FUNCTION_BLOCK PnpXYCalculatorBA (* Composite Function Block Type *)
  (* Standard: 61499-2 *)
  (* Version 0.2, 2003-12-05, JHC, Rockwell Automation, Renamed from NEWCOMPFB. *)
  (* Version 0.1, 2002-01-08, JHC, Rockwell Automation, Added DLY FB as example. *)
  (* Version 0.0, 2000-05-27, JHC, Rockwell Automation *)
  (* Compiler header: package fb.rt.pnp; *)
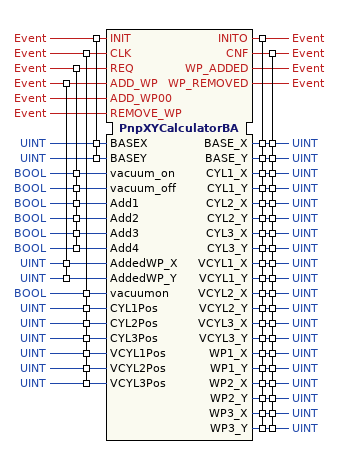
  EVENT_INPUT
    INIT WITH BASEX, BASEY; (* Initialization Request *)
    CLK WITH vacuumon, CYL1Pos, CYL2Pos, CYL3Pos, VCYL1Pos, VCYL2Pos, VCYL3Pos; (* Clock *)
    REQ WITH vacuum_on, vacuum_off, Add1, Add2, Add3, Add4;
    ADD_WP WITH AddedWP_X, AddedWP_Y;
    ADD_WP00;
    REMOVE_WP;
  END_EVENT
  EVENT_OUTPUT
    INITO WITH CYL1_X, CYL1_Y, BASE_Y, BASE_X, CYL2_X, CYL2_Y, VCYL1_X, VCYL1_Y, WP1_X, WP1_Y, WP2_X, WP2_Y, WP3_X, WP3_Y, CYL3_X, CYL3_Y, VCYL2_X, VCYL2_Y, VCYL3_X, VCYL3_Y; (* Initialization Confirm *)
    CNF WITH CYL1_X, CYL1_Y, BASE_Y, BASE_X, CYL2_X, CYL2_Y, VCYL1_X, VCYL1_Y, WP1_X, WP1_Y, WP2_X, WP2_Y, WP3_X, WP3_Y, CYL3_X, CYL3_Y, VCYL2_X, VCYL2_Y, VCYL3_X, VCYL3_Y;
    WP_ADDED;
    WP_REMOVED;
  END_EVENT
  VAR_INPUT
    BASEX : UINT;
    BASEY : UINT;
    vacuum_on : BOOL;
    vacuum_off : BOOL;
    Add1 : BOOL;
    Add2 : BOOL;
    Add3 : BOOL;
    Add4 : BOOL;
    AddedWP_X : UINT;
    AddedWP_Y : UINT;
    vacuumon : BOOL;
    CYL1Pos : UINT;
    CYL2Pos : UINT;
    CYL3Pos : UINT;
    VCYL1Pos : UINT;
    VCYL2Pos : UINT;
    VCYL3Pos : UINT;
  END_VAR
  VAR_OUTPUT
    BASE_X : UINT; (* Response Data from Socket *)
    BASE_Y : UINT; (* Response Data from Socket *)
    CYL1_X : UINT; (* Response Data from Socket *)
    CYL1_Y : UINT; (* Response Data from Socket *)
    CYL2_X : UINT; (* Response Data from Socket *)
    CYL2_Y : UINT; (* Response Data from Socket *)
    CYL3_X : UINT; (* Response Data from Socket *)
    CYL3_Y : UINT; (* Response Data from Socket *)
    VCYL1_X : UINT; (* Response Data from Socket *)
    VCYL1_Y : UINT; (* Response Data from Socket *)
    VCYL2_X : UINT; (* Response Data from Socket *)
    VCYL2_Y : UINT; (* Response Data from Socket *)
    VCYL3_X : UINT; (* Response Data from Socket *)
    VCYL3_Y : UINT; (* Response Data from Socket *)
    WP1_X : UINT; (* Response Data from Socket *)
    WP1_Y : UINT; (* Response Data from Socket *)
    WP2_X : UINT; (* Response Data from Socket *)
    WP2_Y : UINT; (* Response Data from Socket *)
    WP3_X : UINT; (* Response Data from Socket *)
    WP3_Y : UINT; (* Response Data from Socket *)
  END_VAR
  VAR
    cyl1x : UINT;
    cyl2x : UINT;
    cyl3x : UINT;
    vcyl1y : UINT;
    vcyl2y : UINT;
    vcyl3y : UINT;
    wp1x : UINT;
    wp1y : UINT;
    wp2x : UINT;
    wp2y : UINT;
    wp3x : UINT;
    wp3y : UINT;
    wp4x : UINT;
    wp4y : UINT;
    slider1 : BOOL;
    slider2 : BOOL;
    slider3 : BOOL;
    slider4 : BOOL;
    wp1on : BOOL;
    wp2on : BOOL;
    wp3on : BOOL;
    wp4on : BOOL;
  END_VAR
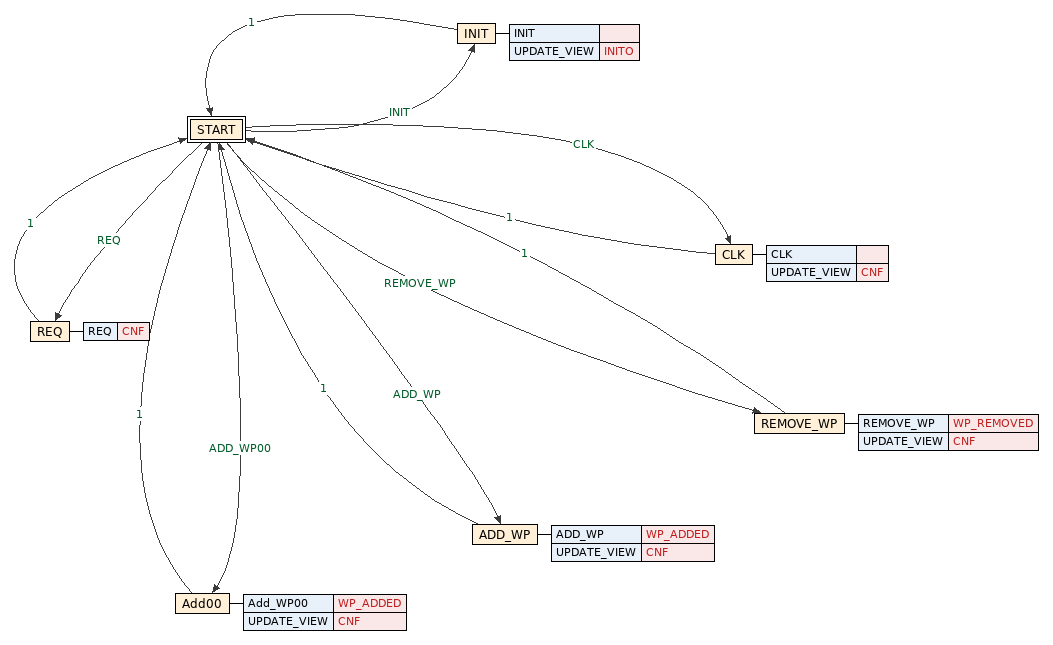
  EC_STATES
    START; (* Initial State *)
    INIT : INIT, UPDATE_VIEW -> INITO; (* Initialization *)
    REQ : REQ -> CNF; (* Normal execution *)
    CLK : CLK, UPDATE_VIEW -> CNF;
    ADD_WP : ADD_WP -> WP_ADDED, UPDATE_VIEW -> CNF;
    REMOVE_WP : REMOVE_WP -> WP_REMOVED, UPDATE_VIEW -> CNF;
    Add00 : Add_WP00 -> WP_ADDED, UPDATE_VIEW -> CNF;
  END_STATES
  EC_TRANSITIONS
    START TO INIT := INIT;
    INIT TO START := 1;
    START TO REQ := REQ;
    REQ TO START := 1;
    START TO CLK := CLK;
    CLK TO START := 1;
    START TO ADD_WP := ADD_WP;
    ADD_WP TO START := 1;
    START TO REMOVE_WP := REMOVE_WP;
    REMOVE_WP TO START := 1;
    START TO Add00 := ADD_WP00;
    Add00 TO START := 1;
  END_TRANSITIONS
  ALGORITHM INIT IN Java: (* Initialization algorithm *)
wp1x.value = 6000;
wp1y.value = 6000;
wp2x.value = 6000;
wp2y.value = 6000;
wp3x.value = 6000;
wp3y.value = 6000;
wp1on.value = false;
wp2on.value = false;
wp3on.value = false;

BASE_X.value = BASEX.value;
BASE_Y.value = BASEY.value;
CYL1_Y.value = BASEY.value;
CYL2_Y.value = BASEY.value;
CYL3_Y.value = BASEY.value;
  END_ALGORITHM
  ALGORITHM REQ IN Java: (* Normally executed algorithm *)

  END_ALGORITHM
  ALGORITHM CLK IN Java:
int cyl1_length = 75;
int cyl2_length = 75;
int cyl3_length = 150;
int vcyl1_length = 75;
int vcyl2_length = 75;
int vcyl3_length = 75;

cyl1x.value = CYL1Pos.value;
cyl2x.value = CYL2Pos.value;
cyl3x.value = CYL3Pos.value;
vcyl1y.value = VCYL1Pos.value;
vcyl2y.value = VCYL2Pos.value;
vcyl3y.value = VCYL3Pos.value;

if(WP1_X.value<=465 && WP1_Y.value>=370){
slider1.value=true;
} else {slider1.value=false;}
if(WP2_X.value<=465 && WP2_Y.value>=370){
slider2.value=true;
} else {slider2.value=false;}
if(WP3_X.value<=465 && WP3_Y.value>=370){
slider3.value=true;
} else {slider3.value=false;}


if (vacuumon.value) {
int vacuumx = VCYL3_X.value;
int vacuumy = VCYL3_Y.value+100;
int dx1 = Math.abs(wp1x.value - vacuumx);
int dy1 = Math.abs(wp1y.value - vacuumy);
int dx2 = Math.abs(wp2x.value - vacuumx);
int dy2 = Math.abs(wp2y.value - vacuumy);
int dx3 = Math.abs(wp3x.value - vacuumx);
int dy3 = Math.abs(wp3y.value - vacuumy);

if (dx1 < 17 && dy1 < 7 && wp2on.value==false && wp3on.value==false){
wp1on.value = true;
}
if (dx2 < 17 && dy2 < 7 && wp1on.value==false && wp3on.value==false){
wp2on.value = true;
}
if (dx3 < 17 && dy3 < 7 && wp2on.value==false && wp1on.value==false){
wp3on.value = true;
}
//System.out.println("Clocking"+dx1+"-"+dy1);

} else {
wp1on.value = false;
wp2on.value = false;
wp3on.value = false;
}

//System.out.println("Clocking");
  END_ALGORITHM
  ALGORITHM UPDATE_VIEW IN Java:
int bx = BASEX.value;
int by = BASEY.value;
CYL1_X.value = bx+22+cyl1x.value;
CYL2_X.value = CYL1_X.value+90+cyl2x.value;
CYL3_X.value = CYL2_X.value+90+cyl3x.value;

VCYL1_X.value = CYL3_X.value+180;
VCYL2_X.value = CYL3_X.value+180;
VCYL3_X.value = CYL3_X.value+180;
//VCYL1_Y.value = by+vcyl1y.value+15;
VCYL1_Y.value = by+vcyl1y.value;
VCYL2_Y.value = VCYL1_Y.value+90+vcyl2y.value;
VCYL3_Y.value = VCYL2_Y.value+90+vcyl3y.value;

if (wp1on.value){
wp1x.value = VCYL3_X.value;
wp1y.value = VCYL3_Y.value+100;
} else if (slider1.value){


/*if(wp1y.value <= 490) {
wp1y.value = wp1y.value+1;
if (slider2.value && wp2y.value >= 476 && wp1y.value >= 476) {
wp1y.value = wp1y.value-1;
} else if (slider3.value && wp3y.value >= 476 && wp1y.value >= 476) {
wp1y.value = wp1y.value-1;
} else if (slider3.value && slider2.value && wp2y.value >= 462 && wp3y.value >= 462 && wp1y.value >= 460) {
wp1y.value = wp1y.value-1;
}
}*/
wp1y.value = wp1y.value+1;

} else {
//wp1y.value = 385;
}

if (wp2on.value){
wp2x.value = VCYL3_X.value;
wp2y.value = VCYL3_Y.value+100;
} else if (slider2.value){



/*if(wp2y.value <= 490) {

wp2y.value = wp2y.value+1;
if (slider1.value && wp1y.value >= 476 && wp2y.value >= 476) {
wp2y.value = wp2y.value-1;
} else if (slider3.value && wp3y.value >= 476 && wp2y.value >= 476) {
wp2y.value = wp2y.value-1;
} else if (slider3.value && slider1.value && wp1y.value >= 462 && wp3y.value >= 462 && wp2y.value >= 460) {
wp2y.value = wp2y.value-1;
}

}*/
wp2y.value = wp2y.value+1;

} else {
//wp2y.value = 535;
}

if (wp3on.value){
wp3x.value = VCYL3_X.value;
wp3y.value = VCYL3_Y.value+100;
} else if (slider3.value){

/*if(wp3y.value <= 490) {

wp3y.value = wp3y.value+1;
if (slider1.value && wp1y.value >= 476 && wp3y.value >= 476) {
wp3y.value = wp3y.value-1;
} else if (slider2.value && wp2y.value >= 476 && wp3y.value >= 476) {
wp3y.value = wp3y.value-1;
} else if (slider2.value && slider1.value && wp1y.value >= 462 && wp2y.value >= 462 && wp3y.value >= 460) {
wp3y.value = wp3y.value-1;
}

}*/
wp3y.value = wp3y.value+1;


} else {
//wp3y.value = 460;
}



WP1_X.value = wp1x.value;
WP1_Y.value = wp1y.value;
WP2_X.value = wp2x.value;
WP2_Y.value = wp2y.value;
WP3_X.value = wp3x.value;
WP3_Y.value = wp3y.value;

//WP1_X.value = bx+300+wp1x.value;
WP1_Y.value = wp1y.value;
//WP2_X.value = bx+300+wp2x.value;
WP2_Y.value = wp2y.value;
//WP3_X.value = bx+300+wp3x.value;
WP3_Y.value = wp3y.value;


/*if (WP1_X.value == 462 && WP1_Y.value >= 535)
{
    WP1_X.value = 6000;
    WP1_Y.value = 6000;
}
if (WP2_X.value == 462 && WP2_Y.value >= 535)
{
    WP2_X.value = 6000;
    WP2_Y.value = 6000;
}
if (WP3_X.value == 462 && WP3_Y.value >= 535)
{
    WP3_X.value = 6000;
    WP3_Y.value = 6000;
}*/


//System.out.println("C1X = " + CYL1_X + " C2X = " + CYL2_X + " VCX = " + VCYL_X + " VCY = " + VCYL_Y);
  END_ALGORITHM
  ALGORITHM ADD_WP IN Java:
if (Add1.value==true) {
wp1x.value = 537;
wp1y.value = 385;
wp1on.value = false;
}
if (Add2.value==true) {
wp2x.value = 612;
wp2y.value = 535;
wp2on.value = false;
}
if (Add3.value==true) {
wp3x.value = 687;
wp3y.value = 460;
wp3on.value = false;
}
  END_ALGORITHM
  ALGORITHM REMOVE_WP IN Java:
if (Add1.value==true) {
wp1on.value = false;
wp1x.value = 6000;
wp1y.value = 6000;
}
if (Add2.value==true) {
wp2on.value = false;
wp2x.value = 6000;
wp2y.value = 6000;
}
if (Add3.value==true) {
wp3on.value = false;
wp3x.value = 6000;
wp3y.value = 6000;
}
  END_ALGORITHM
  ALGORITHM Add_WP00 IN Java:
if (Add1.value==true) {
wp1x.value = 0;
wp1y.value = 215;
wp1on.value = false;
}
if (Add2.value==true) {
wp2x.value = 0;
wp2y.value = 215;
wp2on.value = false;
}
if (Add3.value==true) {
wp3x.value = 0;
wp3y.value = 215;
wp3on.value = false;
}
if (Add4.value==true) {
wp4x.value = 0;
wp4y.value = 215;
wp4on.value = false;
}
  END_ALGORITHM
END_FUNCTION_BLOCK
